(* IEC 61131-3 sources: CodesysTest/export/Function Blocks/IO, 3 files *)

(* ---- FB_IOLinkBlock.pou.st ---- *)
(*#-#-#-#-#-#-#-#-#-#---Declaration---#-#-#-#-#-#-#-#-#-#-#-#-#*)

{attribute 'FBVisuCreator'}
FUNCTION_BLOCK FINAL FB_IOLinkBlock EXTENDS FB_Murr16PointCFGIO
VAR_INPUT
END_VAR
VAR_OUTPUT
	iIOLinkPort4 : WORD;
	iIOLinkPort5 : WORD;
	iIOLinkPort6 : WORD;
	iIOLinkPort7 : WORD;
END_VAR
VAR
END_VAR
(*#-#-#-#-#-#-#-#-#-#---Implementation---#-#-#-#-#-#-#-#-#-#-#-#-#*)

SUPER^();

iIOLinkPort4 :=  TO_WORD(OSCAT_BASIC.WORD_OF_BYTE(B0 := ptrEIPInputs[3], B1 := ptrEIPInputs[2]));
iIOLinkPort5 :=  TO_WORD(OSCAT_BASIC.WORD_OF_BYTE(B0 := ptrEIPInputs[5], B1 := ptrEIPInputs[4]));
iIOLinkPort6 :=  TO_WORD(OSCAT_BASIC.WORD_OF_BYTE(B0 := ptrEIPInputs[7], B1 := ptrEIPInputs[6]));
iIOLinkPort7 :=  TO_WORD(OSCAT_BASIC.WORD_OF_BYTE(B0 := ptrEIPInputs[9], B1 := ptrEIPInputs[8]));

(* ---- FB_Murr16PointCFGIO.pou.st ---- *)
(*#-#-#-#-#-#-#-#-#-#---Declaration---#-#-#-#-#-#-#-#-#-#-#-#-#*)

{attribute 'FBVisuCreator'}
FUNCTION_BLOCK FB_Murr16PointCFGIO EXTENDS FB_BaseObject
VAR_INPUT
	ptrEIPInputs : POINTER TO BYTE;	// Pointer to starting word of EIP Inputs for the I/O Image
    ptrEIPOutputs : POINTER TO BYTE;	// Pointer to starting word of EIP Outputs for the I/O Image

	oPort0Pin2 : BOOL;
	oPort0Pin4 : BOOL;
	oPort1Pin2 : BOOL;
	oPort1Pin4 : BOOL;
	oPort2Pin2 : BOOL;
	oPort2Pin4 : BOOL;
	oPort3Pin2 : BOOL;
	oPort3Pin4 : BOOL;
	oPort4Pin2 : BOOL;
	oPort4Pin4 : BOOL;
	oPort5Pin2 : BOOL;
	oPort5Pin4 : BOOL;
	oPort6Pin2 : BOOL;
	oPort6Pin4 : BOOL;
	oPort7Pin2 : BOOL;
	oPort7Pin4 : BOOL;
END_VAR
VAR_OUTPUT
	iPort0Pin2 : BOOL;
	iPort0Pin4 : BOOL;
	iPort1Pin2 : BOOL;
	iPort1Pin4 : BOOL;
	iPort2Pin2 : BOOL;
	iPort2Pin4 : BOOL;
	iPort3Pin2 : BOOL;
	iPort3Pin4 : BOOL;
	iPort4Pin2 : BOOL;
	iPort4Pin4 : BOOL;
	iPort5Pin2 : BOOL;
	iPort5Pin4 : BOOL;
	iPort6Pin2 : BOOL;
	iPort6Pin4 : BOOL;
	iPort7Pin2 : BOOL;
	iPort7Pin4 : BOOL;
END_VAR
VAR_IN_OUT
END_VAR
VAR
END_VAR(*#-#-#-#-#-#-#-#-#-#---Implementation---#-#-#-#-#-#-#-#-#-#-#-#-#*)

iPort0Pin2 := ptrEIPInputs[1].0;
iPort0Pin4 := ptrEIPInputs[0].0;
iPort1Pin2 := ptrEIPInputs[1].1;
iPort1Pin4 := ptrEIPInputs[0].1;
iPort2Pin2 := ptrEIPInputs[1].2;
iPort2Pin4 := ptrEIPInputs[0].2;
iPort3Pin2 := ptrEIPInputs[1].3;
iPort3Pin4 := ptrEIPInputs[0].3;
iPort4Pin2 := ptrEIPInputs[1].4;
iPort4Pin4 := ptrEIPInputs[0].4;
iPort5Pin2 := ptrEIPInputs[1].5;
iPort5Pin4 := ptrEIPInputs[0].5;
iPort6Pin2 := ptrEIPInputs[1].6;
iPort6Pin4 := ptrEIPInputs[0].6;
iPort7Pin2 := ptrEIPInputs[1].7;
iPort7Pin4 := ptrEIPInputs[0].7;

ptrEIPOutputs[1].0 := oPort0Pin2;
ptrEIPOutputs[0].0 := oPort0Pin4;
ptrEIPOutputs[1].1 := oPort1Pin2;
ptrEIPOutputs[0].1 := oPort1Pin4;
ptrEIPOutputs[1].2 := oPort2Pin2;
ptrEIPOutputs[0].2 := oPort2Pin4;
ptrEIPOutputs[1].3 := oPort3Pin2;
ptrEIPOutputs[0].3 := oPort3Pin4;
ptrEIPOutputs[1].4 := oPort4Pin2;
ptrEIPOutputs[0].4 := oPort4Pin4;
ptrEIPOutputs[1].5 := oPort5Pin2;
ptrEIPOutputs[0].5 := oPort5Pin4;
ptrEIPOutputs[1].6 := oPort6Pin2;
ptrEIPOutputs[0].6 := oPort6Pin4;
ptrEIPOutputs[1].7 := oPort7Pin2;
ptrEIPOutputs[0].7 := oPort7Pin4;

(* ---- FB_Murr56691_IP20.pou.st ---- *)
(*#-#-#-#-#-#-#-#-#-#---Declaration---#-#-#-#-#-#-#-#-#-#-#-#-#*)

{attribute 'FBVisuCreator'}
FUNCTION_BLOCK FB_Murr56691_IP20 EXTENDS FB_BaseObject
VAR_INPUT
	ptrEIPInputs : POINTER TO BYTE;	// Pointer to starting word of EIP Inputs for the I/O Image
    ptrEIPOutputs : POINTER TO BYTE;	// Pointer to starting word of EIP Outputs for the I/O Image

	oX100 : BOOL;
	oX101 : BOOL;
	oX102 : BOOL;
	oX103 : BOOL;
	oX104 : BOOL;
	oX105 : BOOL;
	oX106 : BOOL;
	oX107 : BOOL;
END_VAR
VAR_OUTPUT

	iX000 : BOOL;
	iX001 : BOOL;
	iX002 : BOOL;
	iX003 : BOOL;
	iX004 : BOOL;
	iX005 : BOOL;
	iX006 : BOOL;
	iX007 : BOOL;

	iX100 : BOOL;
	iX101 : BOOL;
	iX102 : BOOL;
	iX103 : BOOL;
	iX104 : BOOL;
	iX105 : BOOL;
	iX106 : BOOL;
	iX107 : BOOL;
END_VAR
VAR_IN_OUT
END_VAR
VAR
END_VAR(*#-#-#-#-#-#-#-#-#-#---Implementation---#-#-#-#-#-#-#-#-#-#-#-#-#*)

//	Function Block: FB_Murr56691_IP20
//	Description: Abstracts a Murr 56691 IP20 I/O Block
//
//	Created by: Ben Hess
//	Created Date: Friday, October 19, 2018

iX100 := ptrEIPInputs[0].0;
iX101 := ptrEIPInputs[0].1;
iX102 := ptrEIPInputs[0].2;
iX103 := ptrEIPInputs[0].3;
iX104 := ptrEIPInputs[0].4;
iX105 := ptrEIPInputs[0].5;
iX106 := ptrEIPInputs[0].6;
iX107 := ptrEIPInputs[0].7;

iX000 := ptrEIPInputs[1].0;
iX001 := ptrEIPInputs[1].1;
iX002 := ptrEIPInputs[1].2;
iX003 := ptrEIPInputs[1].3;
iX004 := ptrEIPInputs[1].4;
iX005 := ptrEIPInputs[1].5;
iX006 := ptrEIPInputs[1].6;
iX007 := ptrEIPInputs[1].7;

ptrEIPOutputs[0].0 := oX100;
ptrEIPOutputs[0].1 := oX101;
ptrEIPOutputs[0].2 := oX102;
ptrEIPOutputs[0].3 := oX103;
ptrEIPOutputs[0].4 := oX104;
ptrEIPOutputs[0].5 := oX105;
ptrEIPOutputs[0].6 := oX106;
ptrEIPOutputs[0].7 := oX107;
